# EPICS substitutions: ek9000App/Db/EL4008.substitutions
file EL4008.template
{       pattern
        {
                TERMINAL,

        }
        {
        }
}
